// TIA Portal V19 export
VAR_GLOBAL   // PLC tag table "Default tag table_4"
   Tag_1 AT %M0.0 : Bool;
END_VAR
